FUNCTION_BLOCK SPLIT_SIGNED_SINT (* Teilt einen SINT-Wert in 2 einseitige Betragswerte auf: NEG_MAG = MAX(0,-Y), POS_MAG = MAX(0,Y). Sonderfall Y=SINT#-128 (SINT-Minimum): -Y wuerde ueberlaufen (Zweierkomplement, |MIN| > MAX) - in diesem Fall wird NEG_MAG auf SINT#127 (SINT-Maximum) begrenzt (Regelungstechnik: Saettigung statt Ueberlauf/Vorzeichenwechsel). Feuert CNF bei jedem REQ, unabhaengig von Wertaenderung - Event-Deduplizierung erfolgt aussen im Adapter-Wrapper AS_SPLIT_SIGNED ueber je einen E_D_FF_ANY pro Seite. *)
  (* Standard: 61499-2 *)
  (* Version 1.0, 2026-09-11, Franz Höpfinger, Einfacher Value/Event-Baustein ohne Event-Dedup - wird vom Adapter-Wrapper AS_SPLIT_SIGNED mit je einem E_D_FF_ANY pro Seite dedupliziert *)
  PACKAGE adapter::Engineering::splitting::signed;
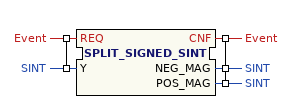
  EVENT_INPUT
    REQ WITH Y; (* Neuer Y-Wert liegt an *)
  END_EVENT
  EVENT_OUTPUT
    CNF WITH NEG_MAG, POS_MAG; (* NEG_MAG/POS_MAG berechnet *)
  END_EVENT
  VAR_INPUT
    Y : SINT; (* Eingangswert *)
  END_VAR
  VAR_OUTPUT
    NEG_MAG : SINT; (* MAX(0, -Y), bei Y=SINT#-128 gesaettigt auf SINT#127 *)
    POS_MAG : SINT; (* MAX(0, Y) *)
  END_VAR
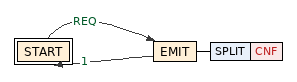
  EC_STATES
    START; (* Initial State *)
    EMIT : SPLIT -> CNF;
  END_STATES
  EC_TRANSITIONS
    START TO EMIT := REQ;
    EMIT TO START := 1;
  END_TRANSITIONS
  ALGORITHM SPLIT IN ST:
IF Y = SINT#-128 THEN
	NEG_MAG := SINT#127;
ELSE
	NEG_MAG := MAX(SINT#0,-Y);
END_IF;
POS_MAG := MAX(SINT#0,Y);
  END_ALGORITHM
END_FUNCTION_BLOCK
